{attribute 'qualified_only'}
VAR_GLOBAL CONSTANT
    // 16 including "Unknown" is the max for an EPICS MBBI/MBBO
    // This is the max number of user-defined states (OUT, TARGET1, YAG...)
    // You can make this smaller if you want to use less memory in your program in exchange for limiting your max state count
    // You can make this larger if you want to use states-based FBs sized beyond the EPICS enum limit
    MAX_STATES: INT := 15;
END_VAR

(* stored: Version 1.1.0.1, ProductVersion 3.1.4022.18
   GVL GeneralConstants: Id {5fbde5e2-29c8-4193-ba17-69759df29f93}, ParameterList True *)
